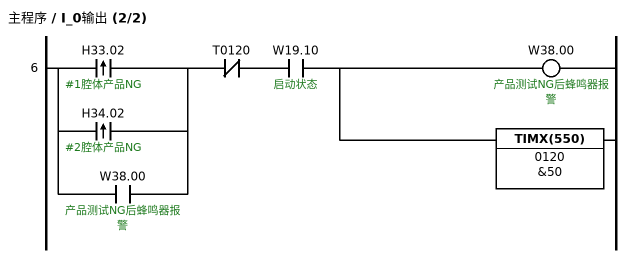
; [picture p48: 主程序 / I_0输出, rungs 6-6]
; rung 6
@LD H33.02  ; #1腔体产品NG
@OR H34.02  ; #2腔体产品NG
OR W38.00  ; 产品测试NG后蜂鸣器报警
ANDNOT T0120
AND W19.10  ; 启动状态
OUT W38.00  ; 产品测试NG后蜂鸣器报警
TIMX(550) 0120 &50

### Section 数据转移

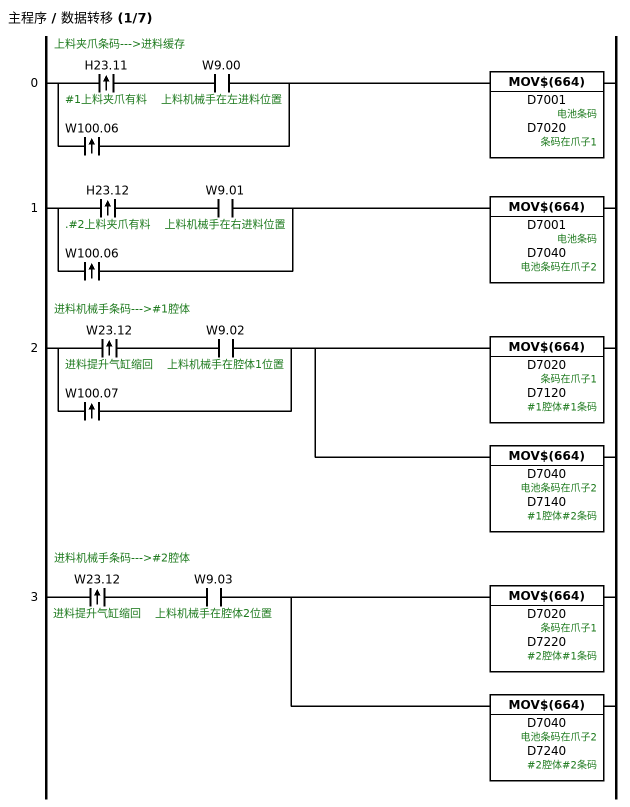
; rung 0: 上料夹爪条码--->进料缓存
@LD H23.11  ; #1上料夹爪有料
AND W9.00  ; 上料机械手在左进料位置
@OR W100.06
MOV$(664) D7001 D7020  ; 电池条码, 条码在爪子1
; rung 1
@LD H23.12  ; .#2上料夹爪有料
AND W9.01  ; 上料机械手在右进料位置
@OR W100.06
MOV$(664) D7001 D7040  ; 电池条码, 电池条码在爪子2
; rung 2: 进料机械手条码--->#1腔体
@LD W23.12  ; 进料提升气缸缩回
AND W9.02  ; 上料机械手在腔体1位置
@OR W100.07
MOV$(664) D7020 D7120  ; 条码在爪子1, #1腔体#1条码
MOV$(664) D7040 D7140  ; 电池条码在爪子2, #1腔体#2条码
; rung 3: 进料机械手条码--->#2腔体
@LD W23.12  ; 进料提升气缸缩回
AND W9.03  ; 上料机械手在腔体2位置
MOV$(664) D7020 D7220  ; 条码在爪子1, #2腔体#1条码
MOV$(664) D7040 D7240  ; 电池条码在爪子2, #2腔体#2条码

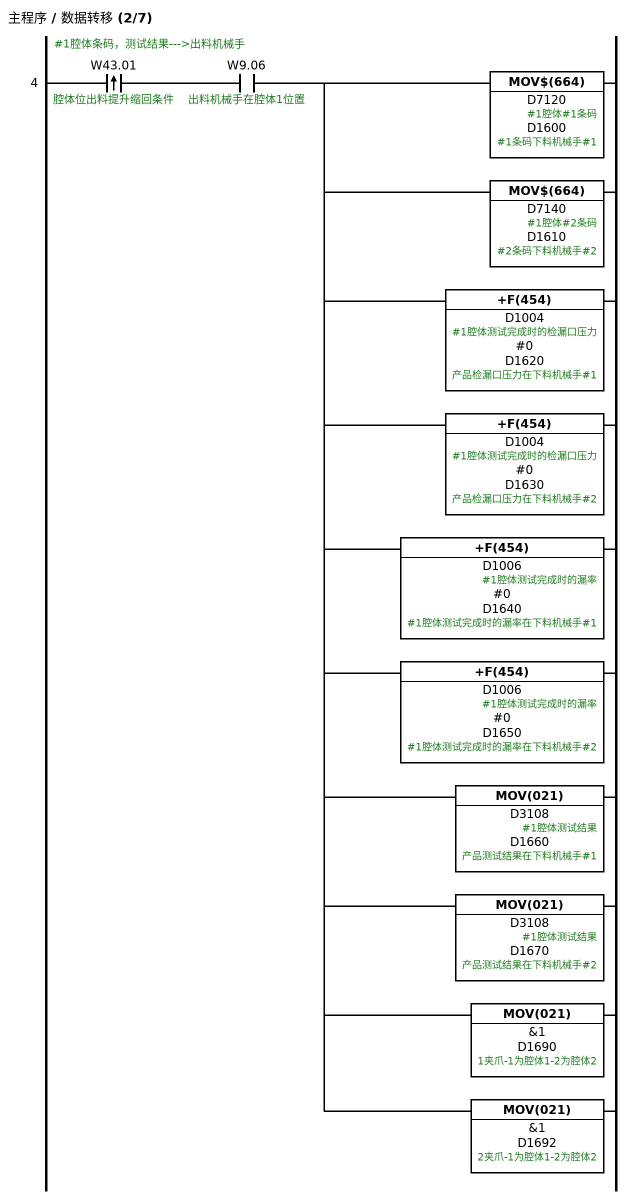
; rung 4: #1腔体条码，测试结果--->出料机械手
@LD W43.01  ; 腔体位出料提升缩回条件
AND W9.06  ; 出料机械手在腔体1位置
MOV$(664) D7120 D1600  ; #1腔体#1条码, #1条码下料机械手#1
MOV$(664) D7140 D1610  ; #1腔体#2条码, #2条码下料机械手#2
+F(454) D1004 #0 D1620  ; #1腔体测试完成时的检漏口压力, 产品检漏口压力在下料机械手#1
+F(454) D1004 #0 D1630  ; #1腔体测试完成时的检漏口压力, 产品检漏口压力在下料机械手#2
+F(454) D1006 #0 D1640  ; #1腔体测试完成时的漏率, #1腔体测试完成时的漏率在下料机械手#1
+F(454) D1006 #0 D1650  ; #1腔体测试完成时的漏率, #1腔体测试完成时的漏率在下料机械手#2
MOV(021) D3108 D1660  ; #1腔体测试结果, 产品测试结果在下料机械手#1
MOV(021) D3108 D1670  ; #1腔体测试结果, 产品测试结果在下料机械手#2
MOV(021) &1 D1690  ; 1夹爪-1为腔体1-2为腔体2
MOV(021) &1 D1692  ; 2夹爪-1为腔体1-2为腔体2

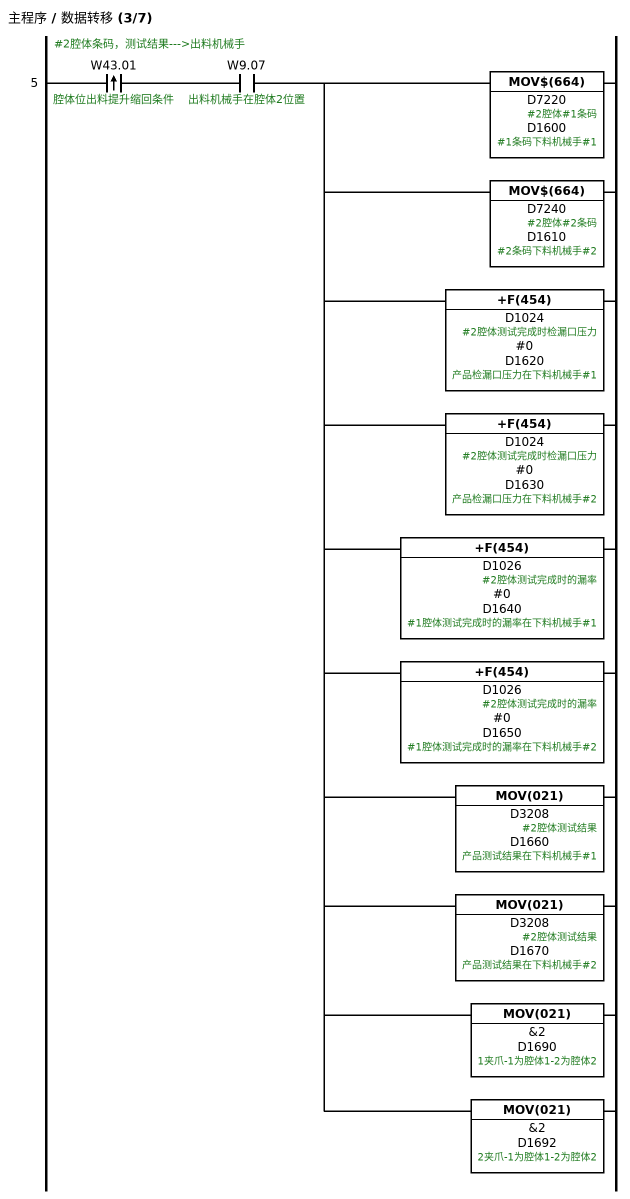
; rung 5: #2腔体条码，测试结果--->出料机械手
@LD W43.01  ; 腔体位出料提升缩回条件
AND W9.07  ; 出料机械手在腔体2位置
MOV$(664) D7220 D1600  ; #2腔体#1条码, #1条码下料机械手#1
MOV$(664) D7240 D1610  ; #2腔体#2条码, #2条码下料机械手#2
+F(454) D1024 #0 D1620  ; #2腔体测试完成时检漏口压力, 产品检漏口压力在下料机械手#1
+F(454) D1024 #0 D1630  ; #2腔体测试完成时检漏口压力, 产品检漏口压力在下料机械手#2
+F(454) D1026 #0 D1640  ; #2腔体测试完成时的漏率, #1腔体测试完成时的漏率在下料机械手#1
+F(454) D1026 #0 D1650  ; #2腔体测试完成时的漏率, #1腔体测试完成时的漏率在下料机械手#2
MOV(021) D3208 D1660  ; #2腔体测试结果, 产品测试结果在下料机械手#1
MOV(021) D3208 D1670  ; #2腔体测试结果, 产品测试结果在下料机械手#2
MOV(021) &2 D1690  ; 1夹爪-1为腔体1-2为腔体2
MOV(021) &2 D1692  ; 2夹爪-1为腔体1-2为腔体2

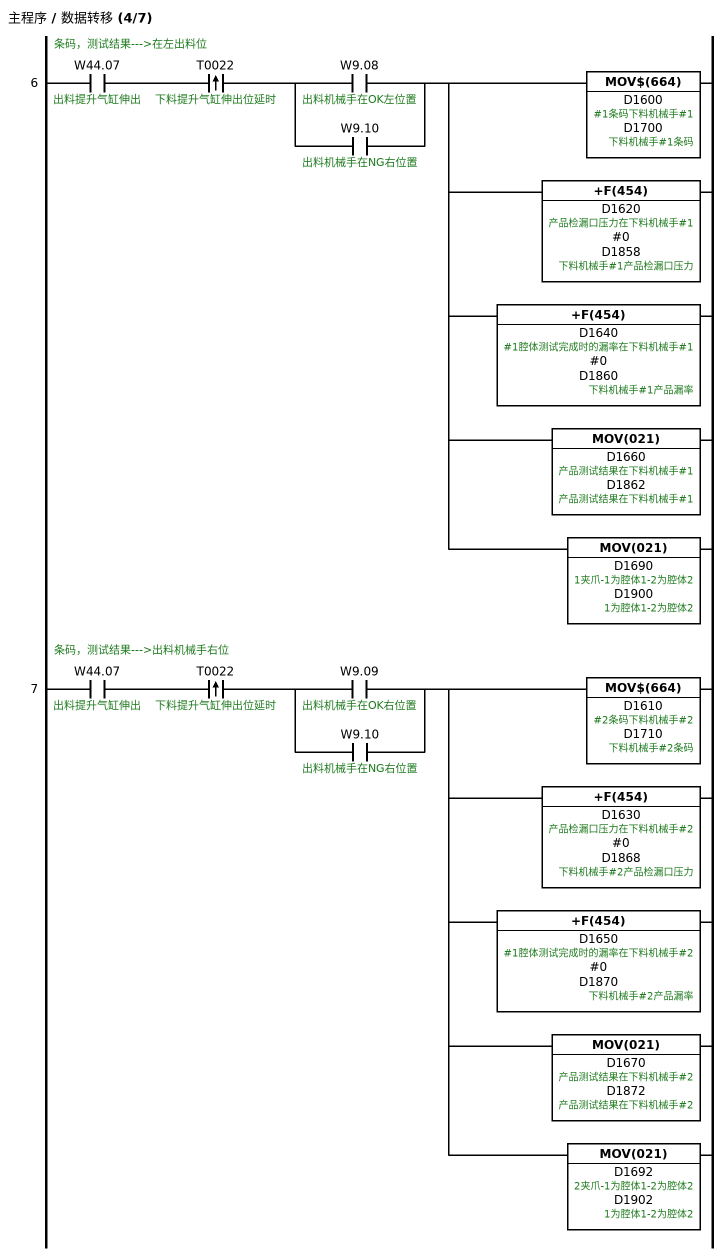
; rung 6: 条码，测试结果--->在左出料位
LD W44.07  ; 出料提升气缸伸出
@AND T0022  ; 下料提升气缸伸出位延时
LD W9.08  ; 出料机械手在OK左位置
OR W9.10  ; 出料机械手在NG右位置
ANDLD
MOV$(664) D1600 D1700  ; #1条码下料机械手#1, 下料机械手#1条码
+F(454) D1620 #0 D1858  ; 产品检漏口压力在下料机械手#1, 下料机械手#1产品检漏口压力
+F(454) D1640 #0 D1860  ; #1腔体测试完成时的漏率在下料机械手#1, 下料机械手#1产品漏率
MOV(021) D1660 D1862  ; 产品测试结果在下料机械手#1
MOV(021) D1690 D1900  ; 1夹爪-1为腔体1-2为腔体2, 1为腔体1-2为腔体2
; rung 7: 条码，测试结果--->出料机械手右位
LD W44.07  ; 出料提升气缸伸出
@AND T0022  ; 下料提升气缸伸出位延时
LD W9.09  ; 出料机械手在OK右位置
OR W9.10  ; 出料机械手在NG右位置
ANDLD
MOV$(664) D1610 D1710  ; #2条码下料机械手#2, 下料机械手#2条码
+F(454) D1630 #0 D1868  ; 产品检漏口压力在下料机械手#2, 下料机械手#2产品检漏口压力
+F(454) D1650 #0 D1870  ; #1腔体测试完成时的漏率在下料机械手#2, 下料机械手#2产品漏率
MOV(021) D1670 D1872  ; 产品测试结果在下料机械手#2
MOV(021) D1692 D1902  ; 2夹爪-1为腔体1-2为腔体2, 1为腔体1-2为腔体2

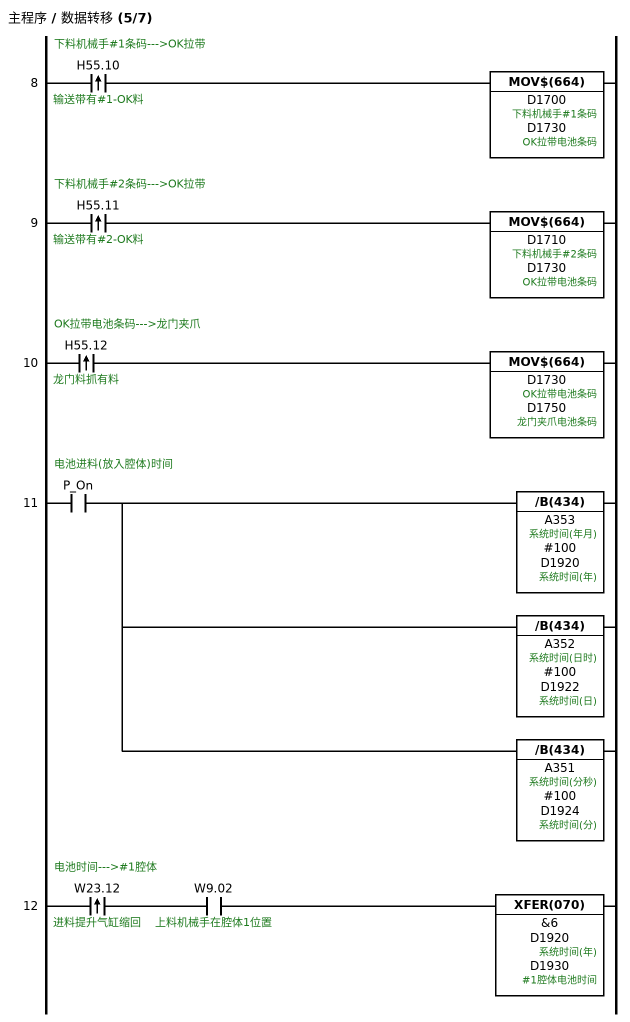
; rung 8: 下料机械手#1条码--->OK拉带
@LD H55.10  ; 输送带有#1-OK料
MOV$(664) D1700 D1730  ; 下料机械手#1条码, OK拉带电池条码
; rung 9: 下料机械手#2条码--->OK拉带
@LD H55.11  ; 输送带有#2-OK料
MOV$(664) D1710 D1730  ; 下料机械手#2条码, OK拉带电池条码
; rung 10: OK拉带电池条码--->龙门夹爪
@LD H55.12  ; 龙门料抓有料
MOV$(664) D1730 D1750  ; OK拉带电池条码, 龙门夹爪电池条码
; rung 11: 电池进料(放入腔体)时间
LD P_On
/B(434) A353 #100 D1920  ; 系统时间(年月), 系统时间(年)
/B(434) A352 #100 D1922  ; 系统时间(日时), 系统时间(日)
/B(434) A351 #100 D1924  ; 系统时间(分秒), 系统时间(分)
; rung 12: 电池时间--->#1腔体
@LD W23.12  ; 进料提升气缸缩回
AND W9.02  ; 上料机械手在腔体1位置
XFER(070) &6 D1920 D1930  ; 系统时间(年), #1腔体电池时间

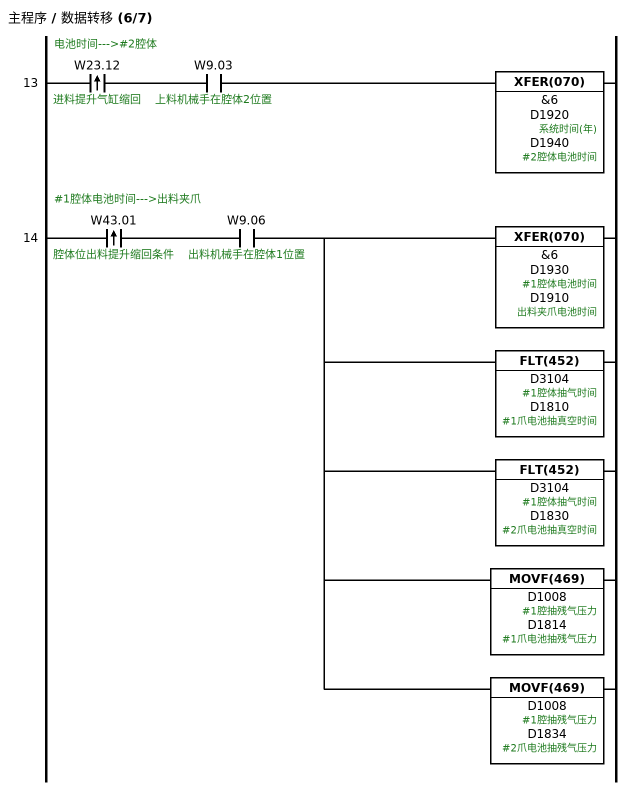
; rung 13: 电池时间--->#2腔体
@LD W23.12  ; 进料提升气缸缩回
AND W9.03  ; 上料机械手在腔体2位置
XFER(070) &6 D1920 D1940  ; 系统时间(年), #2腔体电池时间
; rung 14: #1腔体电池时间--->出料夹爪
@LD W43.01  ; 腔体位出料提升缩回条件
AND W9.06  ; 出料机械手在腔体1位置
XFER(070) &6 D1930 D1910  ; #1腔体电池时间, 出料夹爪电池时间
FLT(452) D3104 D1810  ; #1腔体抽气时间, #1爪电池抽真空时间
FLT(452) D3104 D1830  ; #1腔体抽气时间, #2爪电池抽真空时间
MOVF(469) D1008 D1814  ; #1腔抽残气压力, #1爪电池抽残气压力
MOVF(469) D1008 D1834  ; #1腔抽残气压力, #2爪电池抽残气压力

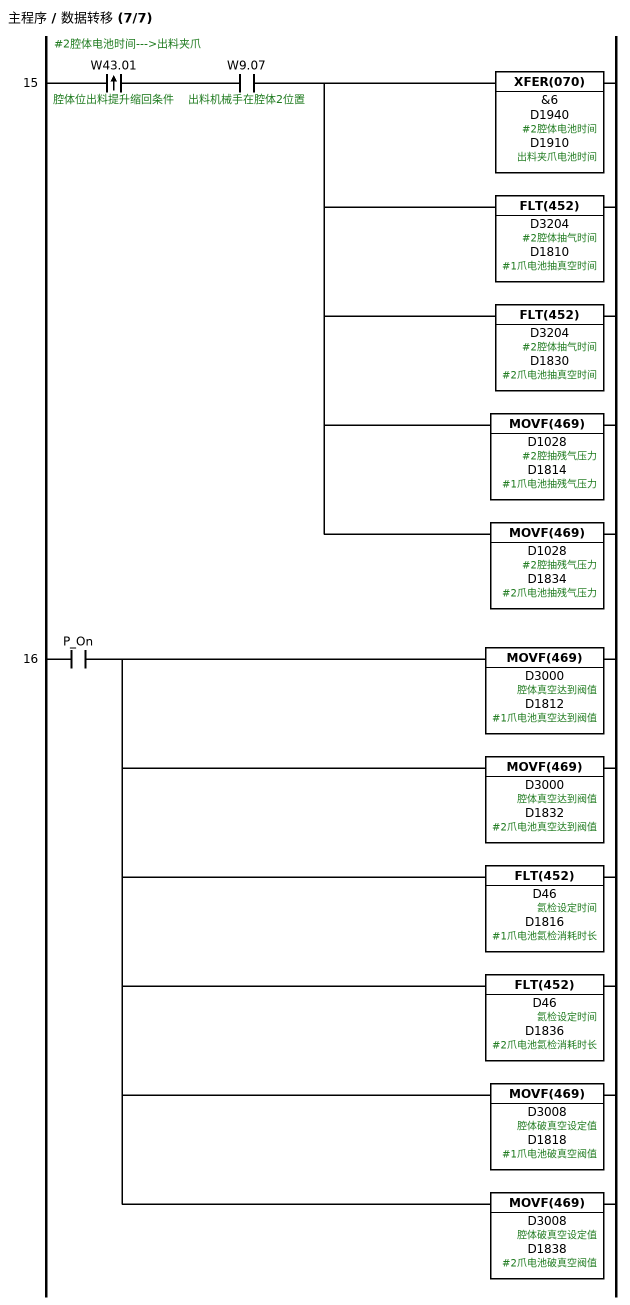
; rung 15: #2腔体电池时间--->出料夹爪
@LD W43.01  ; 腔体位出料提升缩回条件
AND W9.07  ; 出料机械手在腔体2位置
XFER(070) &6 D1940 D1910  ; #2腔体电池时间, 出料夹爪电池时间
FLT(452) D3204 D1810  ; #2腔体抽气时间, #1爪电池抽真空时间
FLT(452) D3204 D1830  ; #2腔体抽气时间, #2爪电池抽真空时间
MOVF(469) D1028 D1814  ; #2腔抽残气压力, #1爪电池抽残气压力
MOVF(469) D1028 D1834  ; #2腔抽残气压力, #2爪电池抽残气压力
; rung 16
LD P_On
MOVF(469) D3000 D1812  ; 腔体真空达到阀值, #1爪电池真空达到阀值
MOVF(469) D3000 D1832  ; 腔体真空达到阀值, #2爪电池真空达到阀值
FLT(452) D46 D1816  ; 氦检设定时间, #1爪电池氦检消耗时长
FLT(452) D46 D1836  ; 氦检设定时间, #2爪电池氦检消耗时长
MOVF(469) D3008 D1818  ; 腔体破真空设定值, #1爪电池破真空阀值
MOVF(469) D3008 D1838  ; 腔体破真空设定值, #2爪电池破真空阀值

### Section 报警

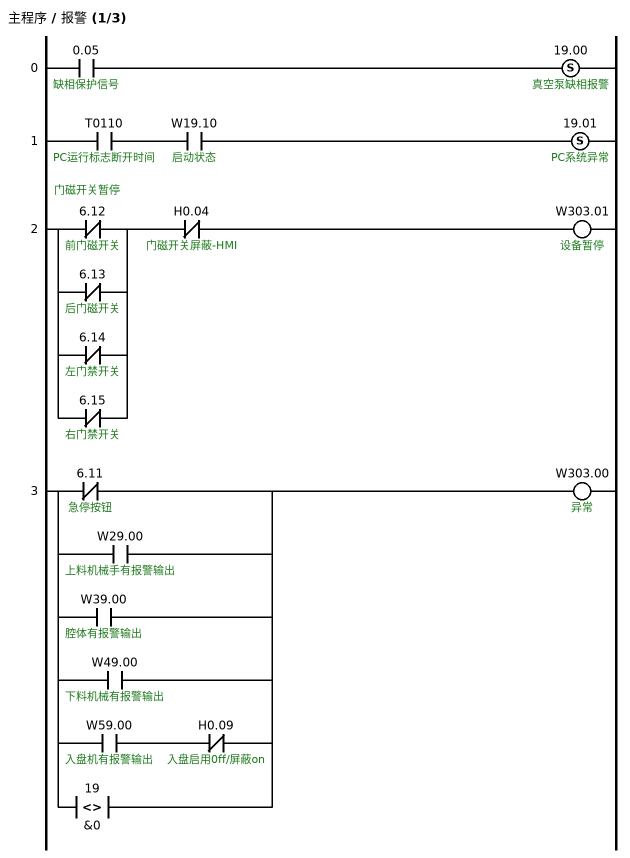
; rung 0
LD 0.05  ; 缺相保护信号
SET 19.00  ; 真空泵缺相报警
; rung 1
LD T0110  ; PC运行标志断开时间
AND W19.10  ; 启动状态
SET 19.01  ; PC系统异常
; rung 2: 门磁开关暂停
LDNOT 6.12  ; 前门磁开关
ORNOT 6.13  ; 后门磁开关
ORNOT 6.14  ; 左门禁开关
ORNOT 6.15  ; 右门禁开关
ANDNOT H0.04  ; 门磁开关屏蔽-HMI
OUT W303.01  ; 设备暂停
; rung 3
LDNOT 6.11  ; 急停按钮
OR W29.00  ; 上料机械手有报警输出
OR W39.00  ; 腔体有报警输出
OR W49.00  ; 下料机械有报警输出
LD W59.00  ; 入盘机有报警输出
ANDNOT H0.09  ; 入盘启用0ff/屏蔽on
ORLD
OR<>(305) 19 &0
OUT W303.00  ; 异常

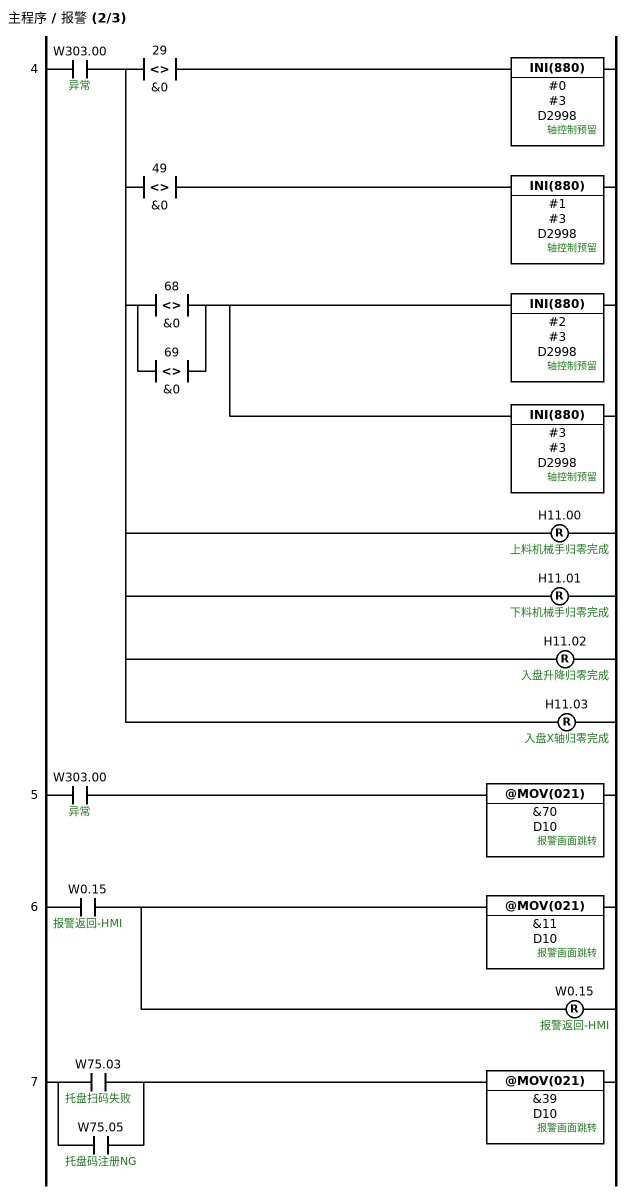
; rung 4
LD W303.00  ; 异常
OUT TR0
AND<>(305) 29 &0
INI(880) #0 #3 D2998  ; 轴控制预留
LD TR0
AND<>(305) 49 &0
INI(880) #1 #3 D2998  ; 轴控制预留
LD TR0
LD<>(305) 68 &0
OR<>(305) 69 &0
ANDLD
INI(880) #2 #3 D2998  ; 轴控制预留
INI(880) #3 #3 D2998  ; 轴控制预留
LD TR0
RSET H11.00  ; 上料机械手归零完成
RSET H11.01  ; 下料机械手归零完成
RSET H11.02  ; 入盘升降归零完成
RSET H11.03  ; 入盘X轴归零完成
; rung 5
LD W303.00  ; 异常
@MOV(021) &70 D10  ; 报警画面跳转
; rung 6
LD W0.15  ; 报警返回-HMI
@MOV(021) &11 D10  ; 报警画面跳转
RSET W0.15  ; 报警返回-HMI
; rung 7
LD W75.03  ; 托盘扫码失败
OR W75.05  ; 托盘码注册NG
@MOV(021) &39 D10  ; 报警画面跳转

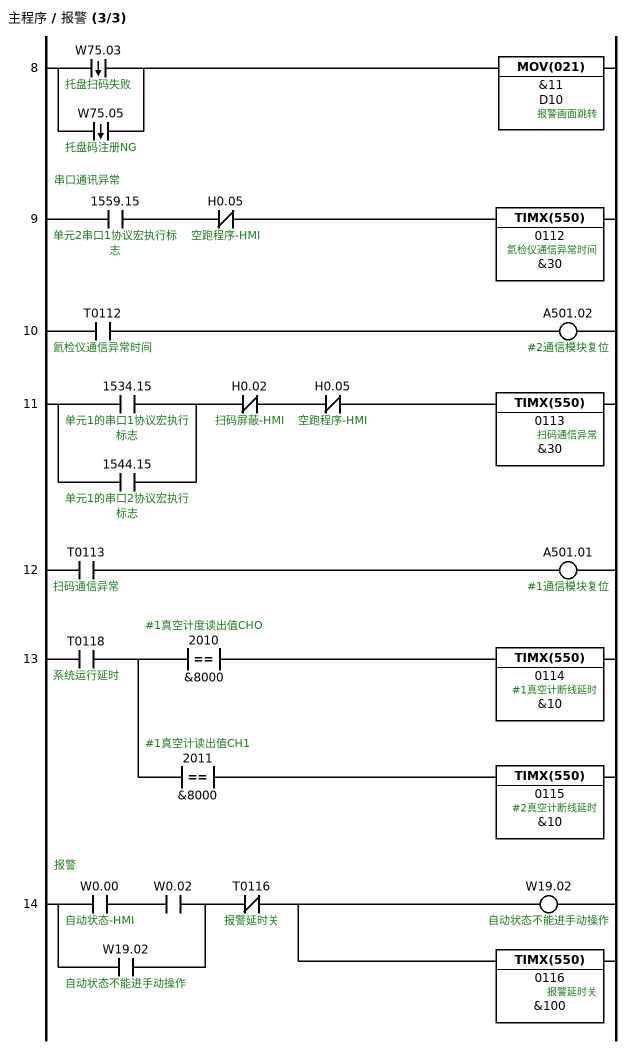
; rung 8
%LD W75.03  ; 托盘扫码失败
%OR W75.05  ; 托盘码注册NG
MOV(021) &11 D10  ; 报警画面跳转
; rung 9: 串口通讯异常
LD 1559.15  ; 单元2串口1协议宏执行标志
ANDNOT H0.05  ; 空跑程序-HMI
TIMX(550) 0112 &30  ; 氦检仪通信异常时间
; rung 10
LD T0112  ; 氦检仪通信异常时间
OUT A501.02  ; #2通信模块复位
; rung 11
LD 1534.15  ; 单元1的串口1协议宏执行标志
OR 1544.15  ; 单元1的串口2协议宏执行标志
ANDNOT H0.02  ; 扫码屏蔽-HMI
ANDNOT H0.05  ; 空跑程序-HMI
TIMX(550) 0113 &30  ; 扫码通信异常
; rung 12
LD T0113  ; 扫码通信异常
OUT A501.01  ; #1通信模块复位
; rung 13
LD T0118  ; 系统运行延时
OUT TR0
AND=(300) 2010 &8000  ; #1真空计度读出值CHO
TIMX(550) 0114 &10  ; #1真空计断线延时
LD TR0
AND=(300) 2011 &8000  ; #1真空计读出值CH1
TIMX(550) 0115 &10  ; #2真空计断线延时
; rung 14: 报警
LD W0.00  ; 自动状态-HMI
AND W0.02
OR W19.02  ; 自动状态不能进手动操作
ANDNOT T0116  ; 报警延时关
OUT W19.02  ; 自动状态不能进手动操作
TIMX(550) 0116 &100  ; 报警延时关

### Section 复位

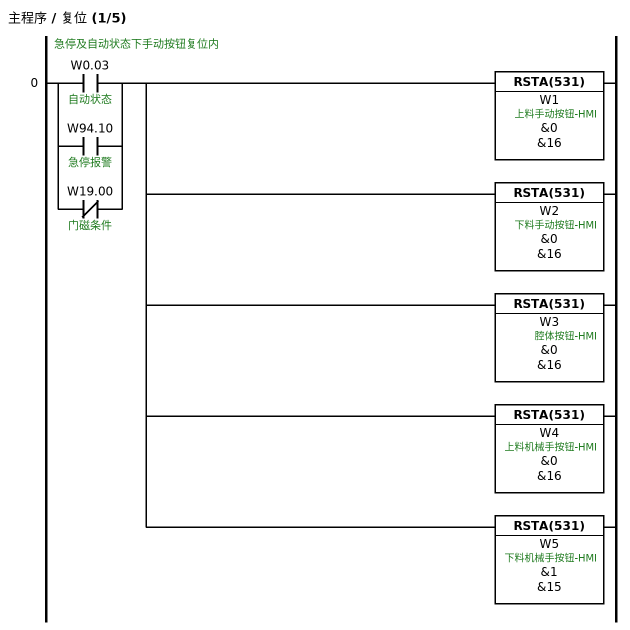
; rung 0: 急停及自动状态下手动按钮复位内
LD W0.03  ; 自动状态
OR W94.10  ; 急停报警
ORNOT W19.00  ; 门磁条件
RSTA(531) W1 &0 &16  ; 上料手动按钮-HMI
RSTA(531) W2 &0 &16  ; 下料手动按钮-HMI
RSTA(531) W3 &0 &16  ; 腔体按钮-HMI
RSTA(531) W4 &0 &16  ; 上料机械手按钮-HMI
RSTA(531) W5 &1 &15  ; 下料机械手按钮-HMI

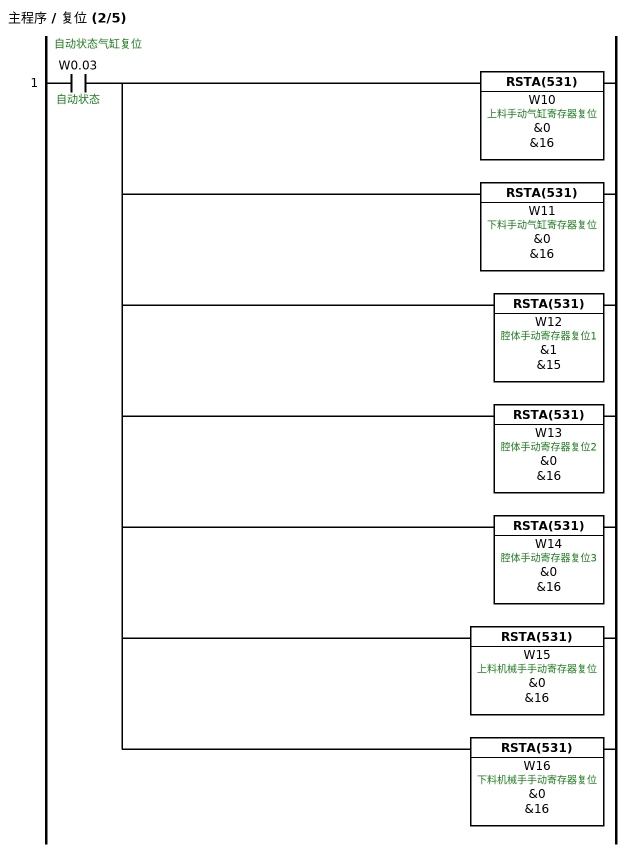
; rung 1: 自动状态气缸复位
LD W0.03  ; 自动状态
RSTA(531) W10 &0 &16  ; 上料手动气缸寄存器复位
RSTA(531) W11 &0 &16  ; 下料手动气缸寄存器复位
RSTA(531) W12 &1 &15  ; 腔体手动寄存器复位1
RSTA(531) W13 &0 &16  ; 腔体手动寄存器复位2
RSTA(531) W14 &0 &16  ; 腔体手动寄存器复位3
RSTA(531) W15 &0 &16  ; 上料机械手手动寄存器复位
RSTA(531) W16 &0 &16  ; 下料机械手手动寄存器复位

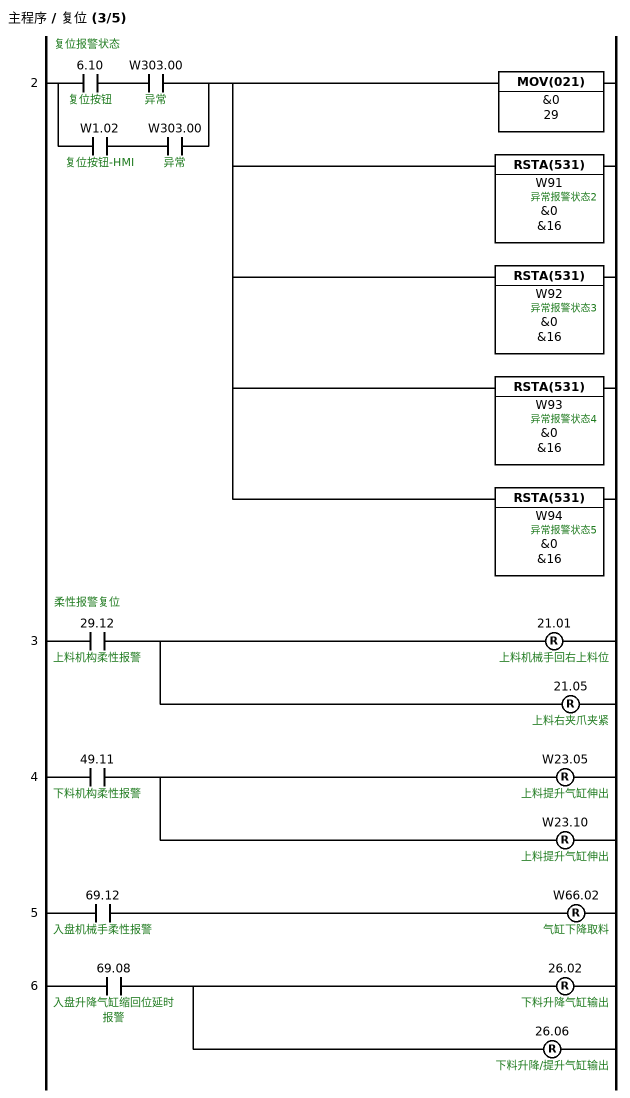
; rung 2: 复位报警状态
LD 6.10  ; 复位按钮
AND W303.00  ; 异常
LD W1.02  ; 复位按钮-HMI
AND W303.00  ; 异常
ORLD
MOV(021) &0 29
RSTA(531) W91 &0 &16  ; 异常报警状态2
RSTA(531) W92 &0 &16  ; 异常报警状态3
RSTA(531) W93 &0 &16  ; 异常报警状态4
RSTA(531) W94 &0 &16  ; 异常报警状态5
; rung 3: 柔性报警复位
LD 29.12  ; 上料机构柔性报警
RSET 21.01  ; 上料机械手回右上料位
RSET 21.05  ; 上料右夹爪夹紧
; rung 4
LD 49.11  ; 下料机构柔性报警
RSET W23.05  ; 上料提升气缸伸出
RSET W23.10  ; 上料提升气缸伸出
; rung 5
LD 69.12  ; 入盘机械手柔性报警
RSET W66.02  ; 气缸下降取料
; rung 6
LD 69.08  ; 入盘升降气缸缩回位延时报警
RSET 26.02  ; 下料升降气缸输出
RSET 26.06  ; 下料升降/提升气缸输出

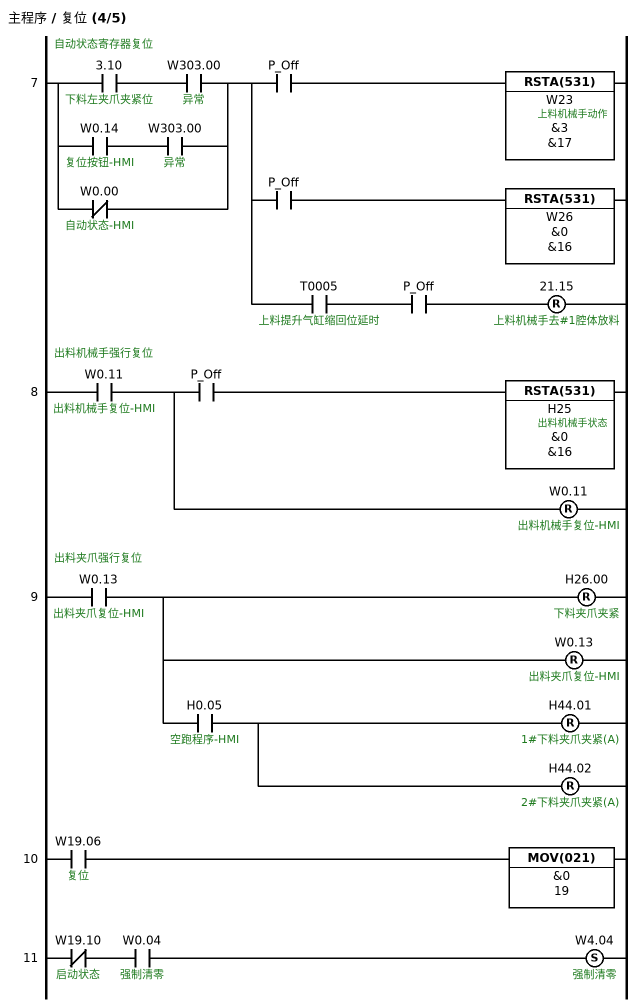
; rung 7: 自动状态寄存器复位
LD 3.10  ; 下料左夹爪夹紧位
AND W303.00  ; 异常
LD W0.14  ; 复位按钮-HMI
AND W303.00  ; 异常
ORLD
ORNOT W0.00  ; 自动状态-HMI
OUT TR0
AND P_Off
RSTA(531) W23 &3 &17  ; 上料机械手动作
LD TR0
AND P_Off
RSTA(531) W26 &0 &16
LD TR0
AND T0005  ; 上料提升气缸缩回位延时
AND P_Off
RSET 21.15  ; 上料机械手去#1腔体放料
; rung 8: 出料机械手强行复位
LD W0.11  ; 出料机械手复位-HMI
OUT TR0
AND P_Off
RSTA(531) H25 &0 &16  ; 出料机械手状态
LD TR0
RSET W0.11  ; 出料机械手复位-HMI
; rung 9: 出料夹爪强行复位
LD W0.13  ; 出料夹爪复位-HMI
RSET H26.00  ; 下料夹爪夹紧
RSET W0.13  ; 出料夹爪复位-HMI
AND H0.05  ; 空跑程序-HMI
RSET H44.01  ; 1#下料夹爪夹紧(A)
RSET H44.02  ; 2#下料夹爪夹紧(A)
; rung 10
LD W19.06  ; 复位
MOV(021) &0 19
; rung 11
LDNOT W19.10  ; 启动状态
AND W0.04  ; 强制清零
SET W4.04  ; 强制清零

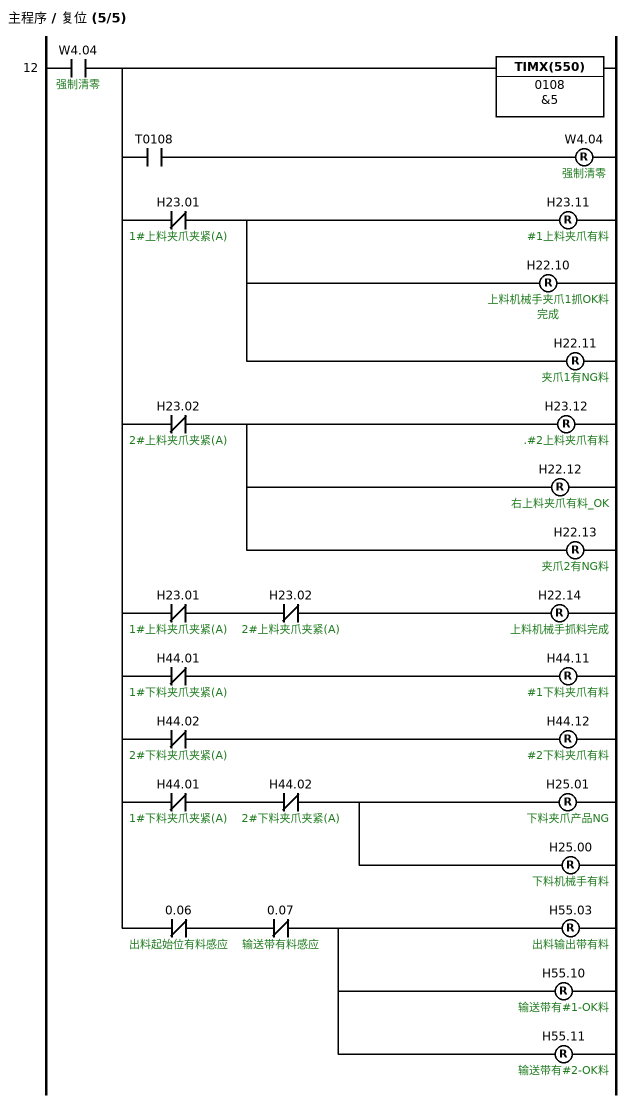
; rung 12
LD W4.04  ; 强制清零
OUT TR0
TIMX(550) 0108 &5
AND T0108
RSET W4.04  ; 强制清零
LD TR0
ANDNOT H23.01  ; 1#上料夹爪夹紧(A)
RSET H23.11  ; #1上料夹爪有料
RSET H22.10  ; 上料机械手夹爪1抓OK料完成
RSET H22.11  ; 夹爪1有NG料
LD TR0
ANDNOT H23.02  ; 2#上料夹爪夹紧(A)
RSET H23.12  ; .#2上料夹爪有料
RSET H22.12  ; 右上料夹爪有料_OK
RSET H22.13  ; 夹爪2有NG料
LD TR0
ANDNOT H23.01  ; 1#上料夹爪夹紧(A)
ANDNOT H23.02  ; 2#上料夹爪夹紧(A)
RSET H22.14  ; 上料机械手抓料完成
LD TR0
ANDNOT H44.01  ; 1#下料夹爪夹紧(A)
RSET H44.11  ; #1下料夹爪有料
LD TR0
ANDNOT H44.02  ; 2#下料夹爪夹紧(A)
RSET H44.12  ; #2下料夹爪有料
LD TR0
ANDNOT H44.01  ; 1#下料夹爪夹紧(A)
ANDNOT H44.02  ; 2#下料夹爪夹紧(A)
RSET H25.01  ; 下料夹爪产品NG
RSET H25.00  ; 下料机械手有料
LD TR0
ANDNOT 0.06  ; 出料起始位有料感应
ANDNOT 0.07  ; 输送带有料感应
RSET H55.03  ; 出料输出带有料
RSET H55.10  ; 输送带有#1-OK料
RSET H55.11  ; 输送带有#2-OK料

### Section END
; rung 0
END(001)

## Program 上料_扫码 (cyclic task 1)

### Section 来料扫码手动

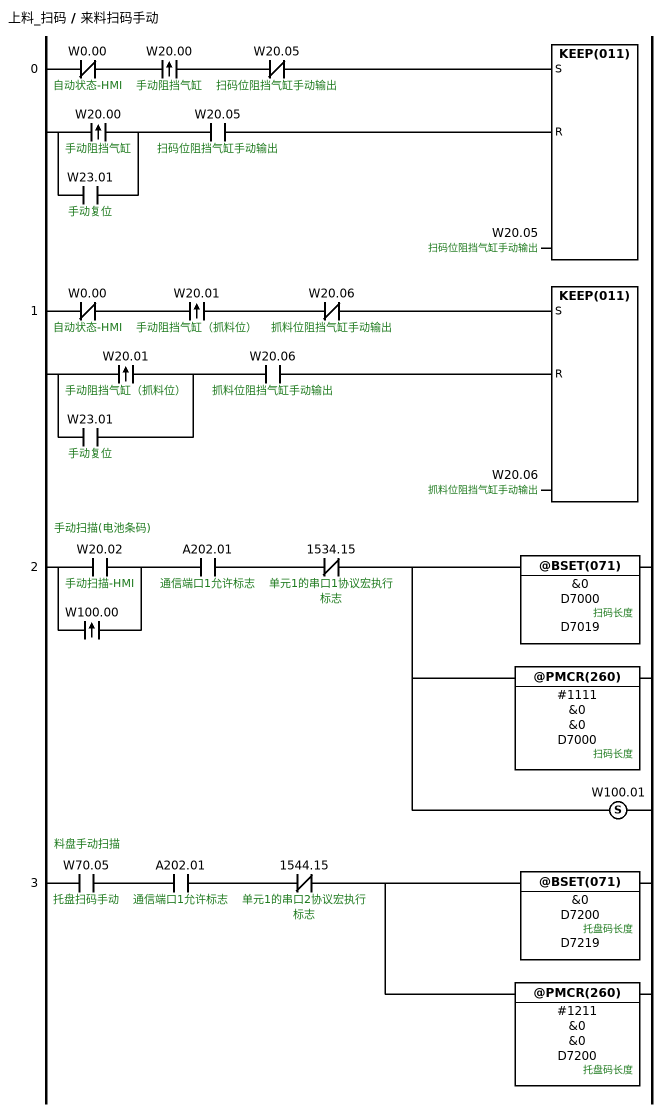
; rung 0
LDNOT W0.00  ; 自动状态-HMI
@AND W20.00  ; 手动阻挡气缸
ANDNOT W20.05  ; 扫码位阻挡气缸手动输出
@LD W20.00  ; 手动阻挡气缸
OR W23.01  ; 手动复位
AND W20.05  ; 扫码位阻挡气缸手动输出
KEEP(011) W20.05  ; 扫码位阻挡气缸手动输出
; rung 1
LDNOT W0.00  ; 自动状态-HMI
@AND W20.01  ; 手动阻挡气缸（抓料位）
ANDNOT W20.06  ; 抓料位阻挡气缸手动输出
@LD W20.01  ; 手动阻挡气缸（抓料位）
OR W23.01  ; 手动复位
AND W20.06  ; 抓料位阻挡气缸手动输出
KEEP(011) W20.06  ; 抓料位阻挡气缸手动输出
; rung 2: 手动扫描(电池条码)
LD W20.02  ; 手动扫描-HMI
@OR W100.00
AND A202.01  ; 通信端口1允许标志
ANDNOT 1534.15  ; 单元1的串口1协议宏执行标志
@BSET(071) &0 D7000 D7019  ; 扫码长度
@PMCR(260) #1111 &0 &0 D7000  ; 扫码长度
SET W100.01
; rung 3: 料盘手动扫描
LD W70.05  ; 托盘扫码手动
AND A202.01  ; 通信端口1允许标志
ANDNOT 1544.15  ; 单元1的串口2协议宏执行标志
@BSET(071) &0 D7200 D7219  ; 托盘码长度
@PMCR(260) #1211 &0 &0 D7200  ; 托盘码长度

### Section 来料扫码自动

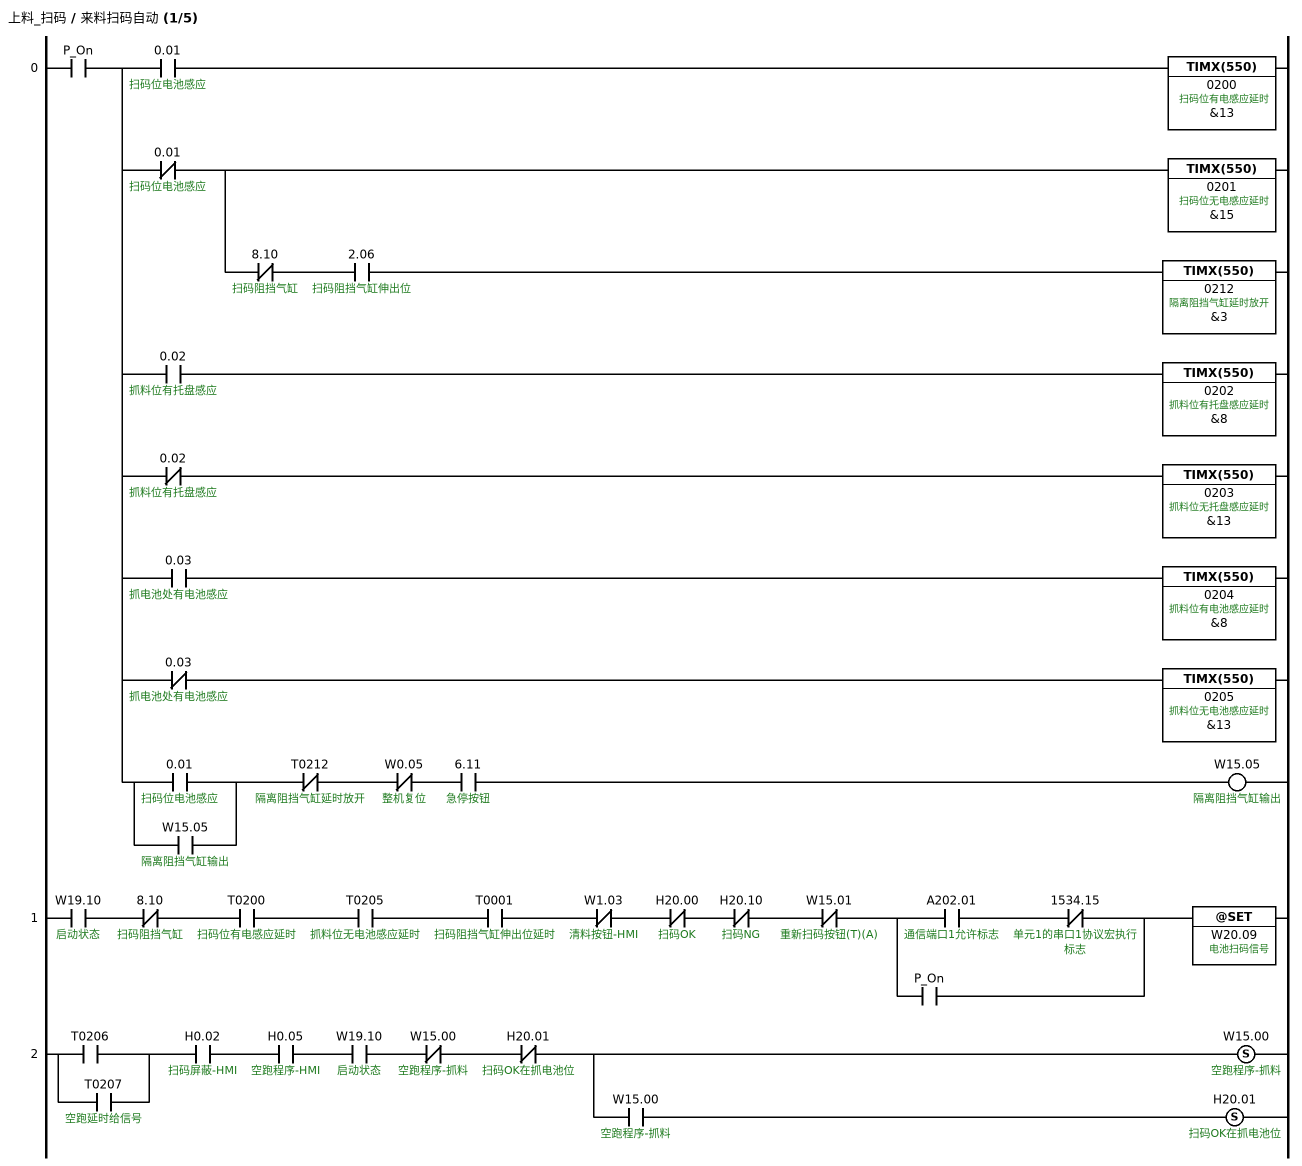
; rung 0
LD P_On
OUT TR0
AND 0.01  ; 扫码位电池感应
TIMX(550) 0200 &13  ; 扫码位有电感应延时
LD TR0
ANDNOT 0.01  ; 扫码位电池感应
TIMX(550) 0201 &15  ; 扫码位无电感应延时
ANDNOT 8.10  ; 扫码阻挡气缸
AND 2.06  ; 扫码阻挡气缸伸出位
TIMX(550) 0212 &3  ; 隔离阻挡气缸延时放开
LD TR0
AND 0.02  ; 抓料位有托盘感应
TIMX(550) 0202 &8  ; 抓料位有托盘感应延时
LD TR0
ANDNOT 0.02  ; 抓料位有托盘感应
TIMX(550) 0203 &13  ; 抓料位无托盘感应延时
LD TR0
AND 0.03  ; 抓电池处有电池感应
TIMX(550) 0204 &8  ; 抓料位有电池感应延时
LD TR0
ANDNOT 0.03  ; 抓电池处有电池感应
TIMX(550) 0205 &13  ; 抓料位无电池感应延时
LD TR0
LD 0.01  ; 扫码位电池感应
OR W15.05  ; 隔离阻挡气缸输出
ANDLD
ANDNOT T0212  ; 隔离阻挡气缸延时放开
ANDNOT W0.05  ; 整机复位
AND 6.11  ; 急停按钮
OUT W15.05  ; 隔离阻挡气缸输出
; rung 1
LD W19.10  ; 启动状态
ANDNOT 8.10  ; 扫码阻挡气缸
AND T0200  ; 扫码位有电感应延时
AND T0205  ; 抓料位无电池感应延时
AND T0001  ; 扫码阻挡气缸伸出位延时
ANDNOT W1.03  ; 清料按钮-HMI
ANDNOT H20.00  ; 扫码OK
ANDNOT H20.10  ; 扫码NG
ANDNOT W15.01  ; 重新扫码按钮(T)(A)
LD A202.01  ; 通信端口1允许标志
ANDNOT 1534.15  ; 单元1的串口1协议宏执行标志
OR P_On
ANDLD
@SET W20.09  ; 电池扫码信号
; rung 2
LD T0206
OR T0207  ; 空跑延时给信号
AND H0.02  ; 扫码屏蔽-HMI
AND H0.05  ; 空跑程序-HMI
AND W19.10  ; 启动状态
ANDNOT W15.00  ; 空跑程序-抓料
ANDNOT H20.01  ; 扫码OK在抓电池位
SET W15.00  ; 空跑程序-抓料
AND W15.00  ; 空跑程序-抓料
SET H20.01  ; 扫码OK在抓电池位

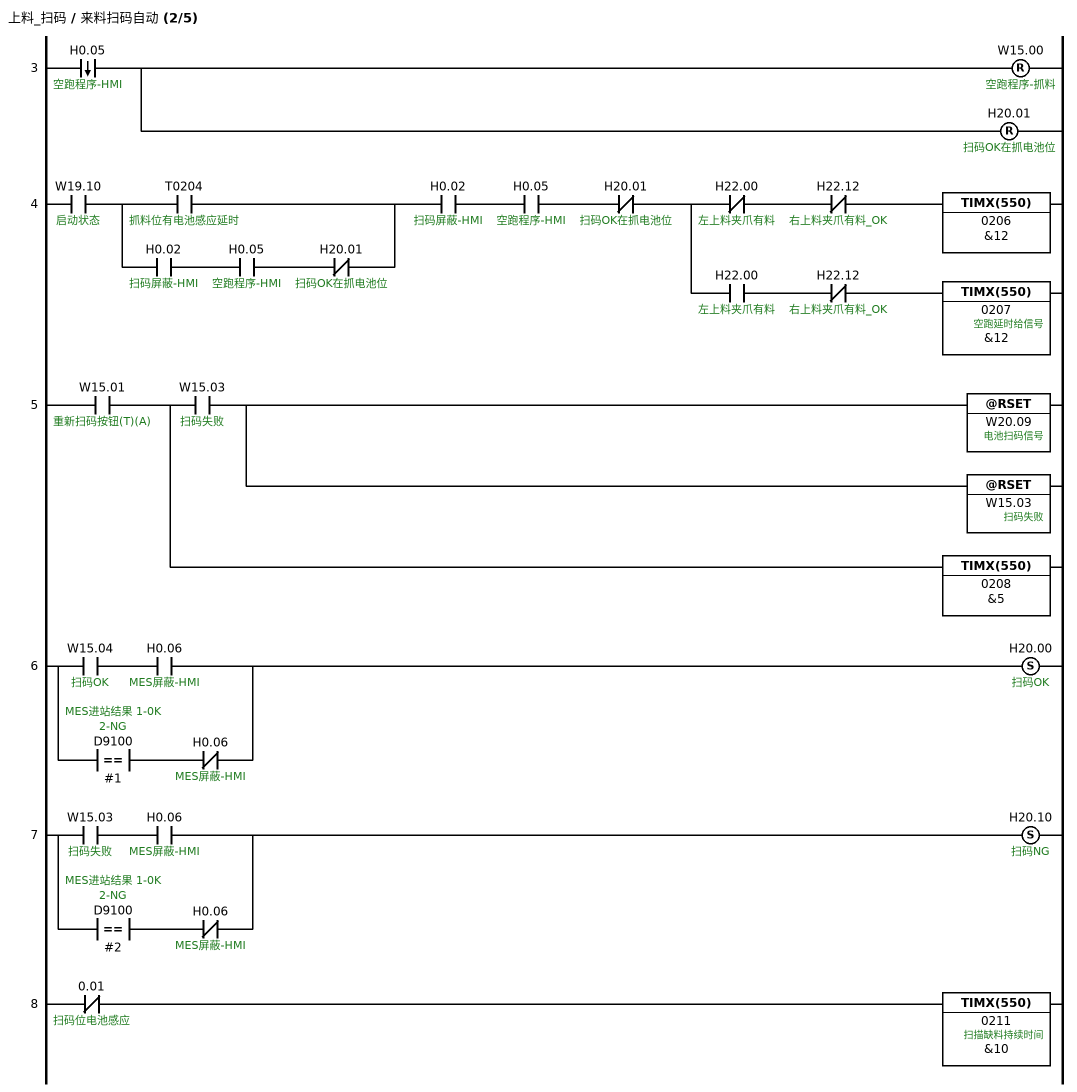
; rung 3
%LD H0.05  ; 空跑程序-HMI
RSET W15.00  ; 空跑程序-抓料
RSET H20.01  ; 扫码OK在抓电池位
; rung 4
LD W19.10  ; 启动状态
LD T0204  ; 抓料位有电池感应延时
LD H0.02  ; 扫码屏蔽-HMI
AND H0.05  ; 空跑程序-HMI
ANDNOT H20.01  ; 扫码OK在抓电池位
ORLD
ANDLD
AND H0.02  ; 扫码屏蔽-HMI
AND H0.05  ; 空跑程序-HMI
ANDNOT H20.01  ; 扫码OK在抓电池位
OUT TR0
ANDNOT H22.00  ; 左上料夹爪有料
ANDNOT H22.12  ; 右上料夹爪有料_OK
TIMX(550) 0206 &12
LD TR0
AND H22.00  ; 左上料夹爪有料
ANDNOT H22.12  ; 右上料夹爪有料_OK
TIMX(550) 0207 &12  ; 空跑延时给信号
; rung 5
LD W15.01  ; 重新扫码按钮(T)(A)
OUT TR0
AND W15.03  ; 扫码失败
@RSET W20.09  ; 电池扫码信号
@RSET W15.03  ; 扫码失败
LD TR0
TIMX(550) 0208 &5
; rung 6
LD W15.04  ; 扫码OK
AND H0.06  ; MES屏蔽-HMI
LD=(300) D9100 #1  ; MES进站结果 1-0K 2-NG
ANDNOT H0.06  ; MES屏蔽-HMI
ORLD
SET H20.00  ; 扫码OK
; rung 7
LD W15.03  ; 扫码失败
AND H0.06  ; MES屏蔽-HMI
LD=(300) D9100 #2  ; MES进站结果 1-0K 2-NG
ANDNOT H0.06  ; MES屏蔽-HMI
ORLD
SET H20.10  ; 扫码NG
; rung 8
LDNOT 0.01  ; 扫码位电池感应
TIMX(550) 0211 &10  ; 扫描缺料持续时间

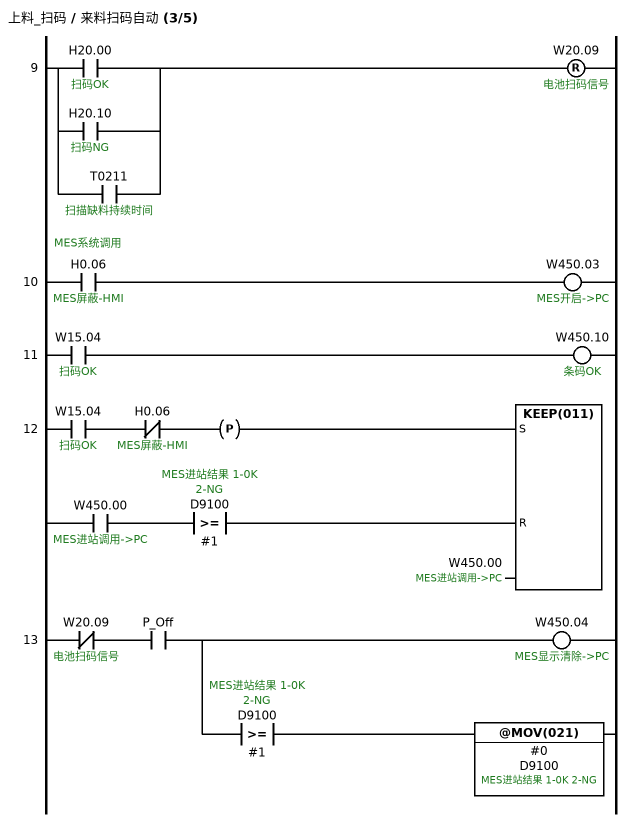
; rung 9
LD H20.00  ; 扫码OK
OR H20.10  ; 扫码NG
OR T0211  ; 扫描缺料持续时间
RSET W20.09  ; 电池扫码信号
; rung 10: MES系统调用
LD H0.06  ; MES屏蔽-HMI
OUT W450.03  ; MES开启->PC
; rung 11
LD W15.04  ; 扫码OK
OUT W450.10  ; 条码OK
; rung 12
LD W15.04  ; 扫码OK
ANDNOT H0.06  ; MES屏蔽-HMI
UP(521)
LD W450.00  ; MES进站调用->PC
AND>=(325) D9100 #1  ; MES进站结果 1-0K 2-NG
KEEP(011) W450.00  ; MES进站调用->PC
; rung 13
LDNOT W20.09  ; 电池扫码信号
AND P_Off
OUT W450.04  ; MES显示清除->PC
AND>=(325) D9100 #1  ; MES进站结果 1-0K 2-NG
@MOV(021) #0 D9100  ; MES进站结果 1-0K 2-NG

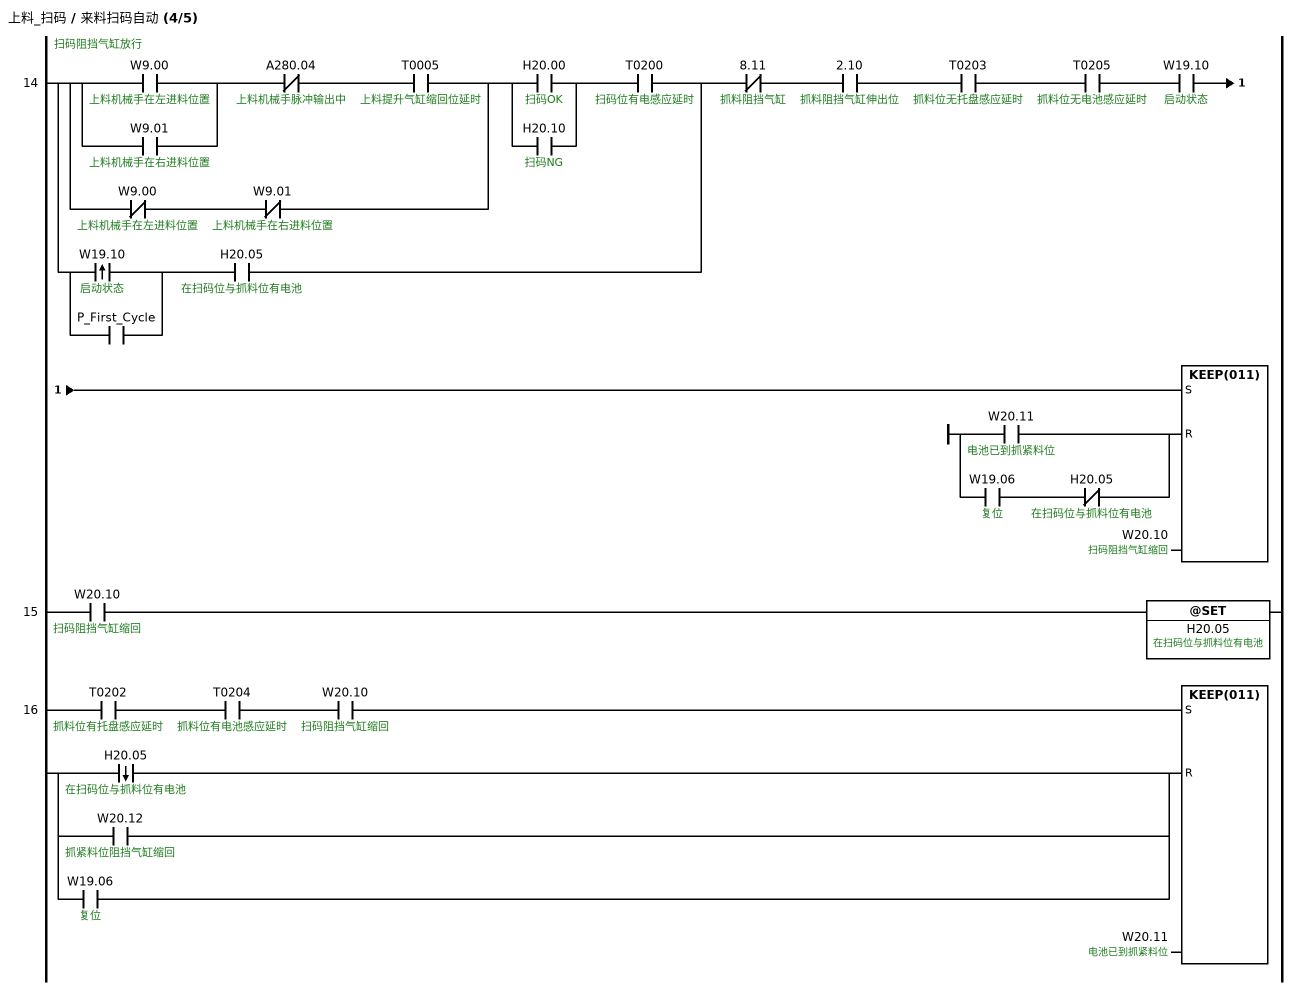
; rung 14: 扫码阻挡气缸放行
LD W9.00  ; 上料机械手在左进料位置
OR W9.01  ; 上料机械手在右进料位置
ANDNOT A280.04  ; 上料机械手脉冲输出中
AND T0005  ; 上料提升气缸缩回位延时
LDNOT W9.00  ; 上料机械手在左进料位置
ANDNOT W9.01  ; 上料机械手在右进料位置
ORLD
LD H20.00  ; 扫码OK
OR H20.10  ; 扫码NG
ANDLD
AND T0200  ; 扫码位有电感应延时
@LD W19.10  ; 启动状态
OR P_First_Cycle
AND H20.05  ; 在扫码位与抓料位有电池
ORLD
ANDNOT 8.11  ; 抓料阻挡气缸
AND 2.10  ; 抓料阻挡气缸伸出位
AND T0203  ; 抓料位无托盘感应延时
AND T0205  ; 抓料位无电池感应延时
AND W19.10  ; 启动状态
LD W20.11  ; 电池已到抓紧料位
LD W19.06  ; 复位
ANDNOT H20.05  ; 在扫码位与抓料位有电池
ORLD
KEEP(011) W20.10  ; 扫码阻挡气缸缩回
; rung 15
LD W20.10  ; 扫码阻挡气缸缩回
@SET H20.05  ; 在扫码位与抓料位有电池
; rung 16
LD T0202  ; 抓料位有托盘感应延时
AND T0204  ; 抓料位有电池感应延时
AND W20.10  ; 扫码阻挡气缸缩回
%LD H20.05  ; 在扫码位与抓料位有电池
OR W20.12  ; 抓紧料位阻挡气缸缩回
OR W19.06  ; 复位
KEEP(011) W20.11  ; 电池已到抓紧料位

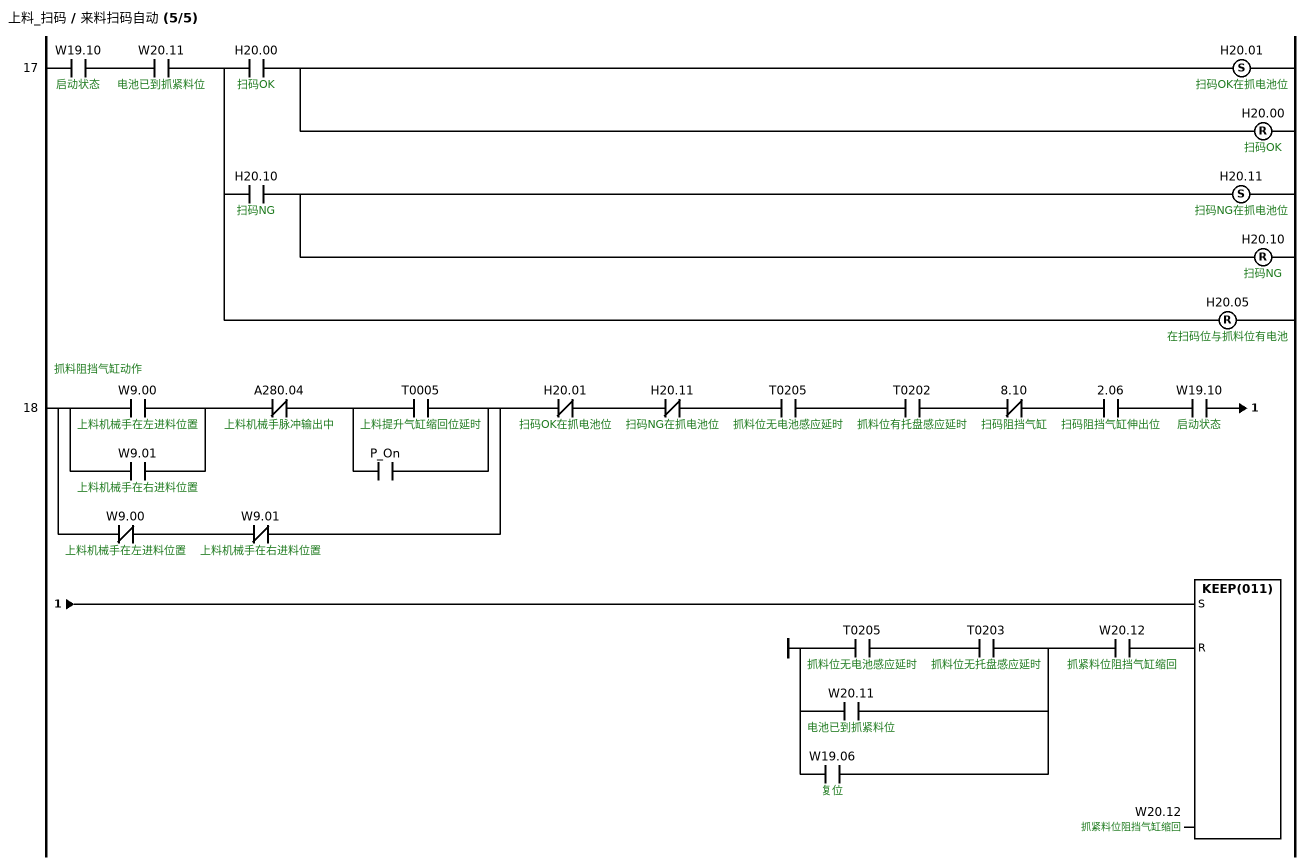
; rung 17
LD W19.10  ; 启动状态
AND W20.11  ; 电池已到抓紧料位
OUT TR0
AND H20.00  ; 扫码OK
SET H20.01  ; 扫码OK在抓电池位
RSET H20.00  ; 扫码OK
LD TR0
AND H20.10  ; 扫码NG
SET H20.11  ; 扫码NG在抓电池位
RSET H20.10  ; 扫码NG
LD TR0
RSET H20.05  ; 在扫码位与抓料位有电池
; rung 18: 抓料阻挡气缸动作
LD W9.00  ; 上料机械手在左进料位置
OR W9.01  ; 上料机械手在右进料位置
ANDNOT A280.04  ; 上料机械手脉冲输出中
LD T0005  ; 上料提升气缸缩回位延时
OR P_On
ANDLD
LDNOT W9.00  ; 上料机械手在左进料位置
ANDNOT W9.01  ; 上料机械手在右进料位置
ORLD
ANDNOT H20.01  ; 扫码OK在抓电池位
ANDNOT H20.11  ; 扫码NG在抓电池位
AND T0205  ; 抓料位无电池感应延时
AND T0202  ; 抓料位有托盘感应延时
ANDNOT 8.10  ; 扫码阻挡气缸
AND 2.06  ; 扫码阻挡气缸伸出位
AND W19.10  ; 启动状态
LD T0205  ; 抓料位无电池感应延时
AND T0203  ; 抓料位无托盘感应延时
OR W20.11  ; 电池已到抓紧料位
OR W19.06  ; 复位
AND W20.12  ; 抓紧料位阻挡气缸缩回
KEEP(011) W20.12  ; 抓紧料位阻挡气缸缩回

### Section 条码读取

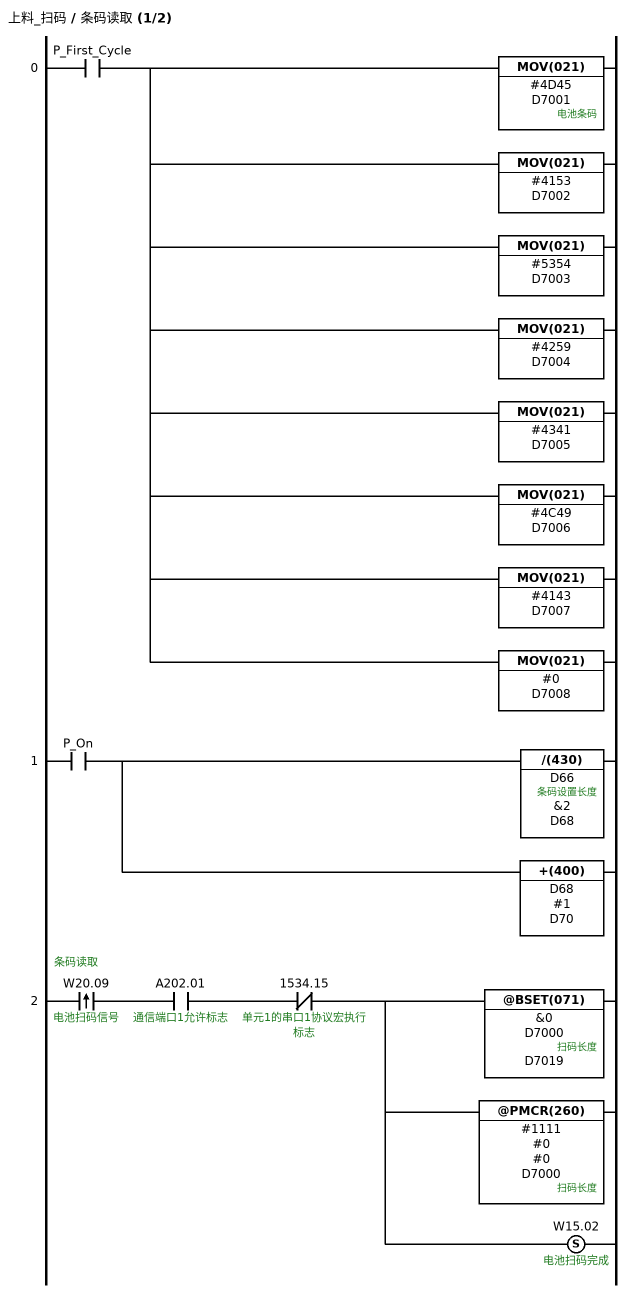
; rung 0
LD P_First_Cycle
MOV(021) #4D45 D7001  ; 电池条码
MOV(021) #4153 D7002
MOV(021) #5354 D7003
MOV(021) #4259 D7004
MOV(021) #4341 D7005
MOV(021) #4C49 D7006
MOV(021) #4143 D7007
MOV(021) #0 D7008
; rung 1
LD P_On
/(430) D66 &2 D68  ; 条码设置长度
+(400) D68 #1 D70
; rung 2: 条码读取
@LD W20.09  ; 电池扫码信号
AND A202.01  ; 通信端口1允许标志
ANDNOT 1534.15  ; 单元1的串口1协议宏执行标志
@BSET(071) &0 D7000 D7019  ; 扫码长度
@PMCR(260) #1111 #0 #0 D7000  ; 扫码长度
SET W15.02  ; 电池扫码完成

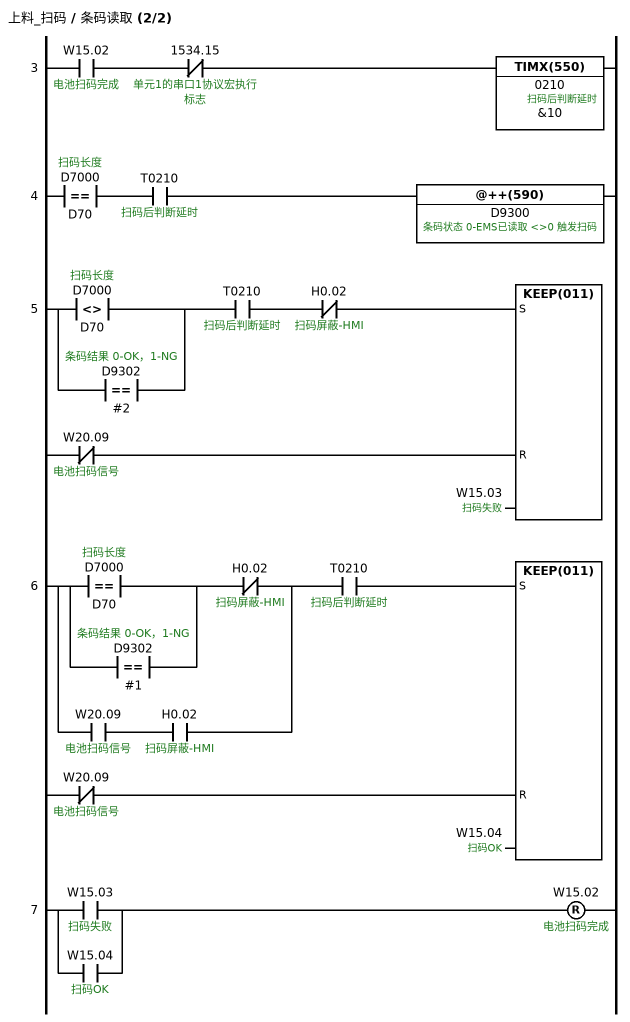
; rung 3
LD W15.02  ; 电池扫码完成
ANDNOT 1534.15  ; 单元1的串口1协议宏执行标志
TIMX(550) 0210 &10  ; 扫码后判断延时
; rung 4
LD=(300) D7000 D70  ; 扫码长度
AND T0210  ; 扫码后判断延时
@++(590) D9300  ; 条码状态 0-EMS已读取 <>0 触发扫码
; rung 5
LD<>(305) D7000 D70  ; 扫码长度
OR=(300) D9302 #2  ; 条码结果 0-OK，1-NG
AND T0210  ; 扫码后判断延时
ANDNOT H0.02  ; 扫码屏蔽-HMI
LDNOT W20.09  ; 电池扫码信号
KEEP(011) W15.03  ; 扫码失败
; rung 6
LD=(300) D7000 D70  ; 扫码长度
OR=(300) D9302 #1  ; 条码结果 0-OK，1-NG
ANDNOT H0.02  ; 扫码屏蔽-HMI
LD W20.09  ; 电池扫码信号
AND H0.02  ; 扫码屏蔽-HMI
ORLD
AND T0210  ; 扫码后判断延时
LDNOT W20.09  ; 电池扫码信号
KEEP(011) W15.04  ; 扫码OK
; rung 7
LD W15.03  ; 扫码失败
OR W15.04  ; 扫码OK
RSET W15.02  ; 电池扫码完成

### Section 输出_报警_复位

